(*
Nazwa:			E_GripperScrewerState
Opis:			Stan zakecarki szczekowej
Wersja:			v0.1
Data:			2018-10-10
Autor:			TW
Urzadzenia:		
Konfiguracja:	
Info:
*)

TYPE E_GripperScrewer :
(	
	
	eReady				:= 1,
	eToPushingPosition	:= 2,
	eToScrewingPosition	:= 3,
	ePushed				:= 4,			
	eFindingScrew		:= 5,			
	eScrewing			:= 6,			
	eGoingUp			:= 7,			
	eDone				:= 8,
	eNotDone			:= 9,
	eHolding			:= 10
	
):= eReady;
END_TYPE

(* stored: Version 1.1.0.1, ProductVersion 3.1.4026.13, FileIdentifier 9883777a6c7776712b839ced737cbdd95e4a012b, FileSignature 37860da4cef58d4caf88446f28a2ba1575ea28685497284d9016905c0282539331a466cc143cc74fa85a8ce2e0fa94308fbd07f7c4dd82918d364ced66e52da523da3d067de6ff0b613bfd1ae457d81756a62d7e5f4c80df315244b4f64d10058826011ebde89f146dee9d0cc0d92ff1144fbb17416cc6b98a0fe17dfecf2a1c12cd674afa137916ea8f61a3760f7c23c4298a08a9731d9d4f1a9b129d4803757eda631c7cf61515023c89faa5f89288f7e99fa0055d0b75610659d10b8d427b2c9a7d8a5c45a6c527d00ce14483ac563c3298ad48f407f9fb4d62c2750e3891370f80cf6e0e379c7899fd6406d6a2b97e4e9bb05743a2ba6f5fc4611d74e1e9
   DUT E_GripperScrewer: Id {dcc13ad1-e2f2-49e5-ae65-1db066c76a92} *)
